Omron CX-Programmer project NewProject (CX-Programmer 9.73)

# PLC NewPLC1: CP1L-E EM

## Global symbols (name address type ; comment)
0.01 BOOL  ; SILINDER MAX (DISTRIBUTION)
0.04 BOOL  ; LIMIT SWITCH KIRI (DISTRIBUTION)
0.05 BOOL  ; LIMIT SWITCH KANAN (DISTRIBUTION)
0.06 BOOL  ; SENSOR BENDA (DISTRIBUTION)
100.00 BOOL  ; SOLENOID (DISTRIBUTION)
100.01 BOOL  ; SUCKER (DISTRIBUTION)
100.02 BOOL  ; BLOW (DISTRIBUTION)
100.03 BOOL  ; MOTOR KIRI (DISTRIBUTION)
100.04 BOOL  ; MOTOR KANAN (DISTRIBUTION)
101.00 BOOL  ; MOTOR KIRI (HANDLING)
101.01 BOOL  ; MOTOR KANAN (HANDLING)
101.02 BOOL  ; SOLENOID (HANDLING)
101.03 BOOL  ; GRAPLE (HANDLING)
101.04 BOOL  ; GRAPLE (HANDLING)
101.07 BOOL  ; TIDAK KIRIM DATA
1.00 BOOL  ; SENSOR BENDA AWAL (HANDLING)
1.01 BOOL  ; LIMIT SWITCH KIRI (HANDLING)
1.02 BOOL  ; LIMIT SWITCH KANAN (HANDLING)
1.03 BOOL  ; LIMIT SWITCH TENGAH (HANDLING)
1.04 BOOL  ; SILINDER MAX (HANDLING)
1.05 BOOL  ; SILINDER MIN (HANDLING)
1.06 BOOL  ; SENSOR BENDA GRAPLE (HANDLING)
W0.00 BOOL  ; START
W0.01 BOOL  ; STOP
W0.02 BOOL  ; RESET
W0.03 BOOL  ; SELECTOR SWITCH

## Program NewProgram1 (cyclic task 0)

### Section CONTROL

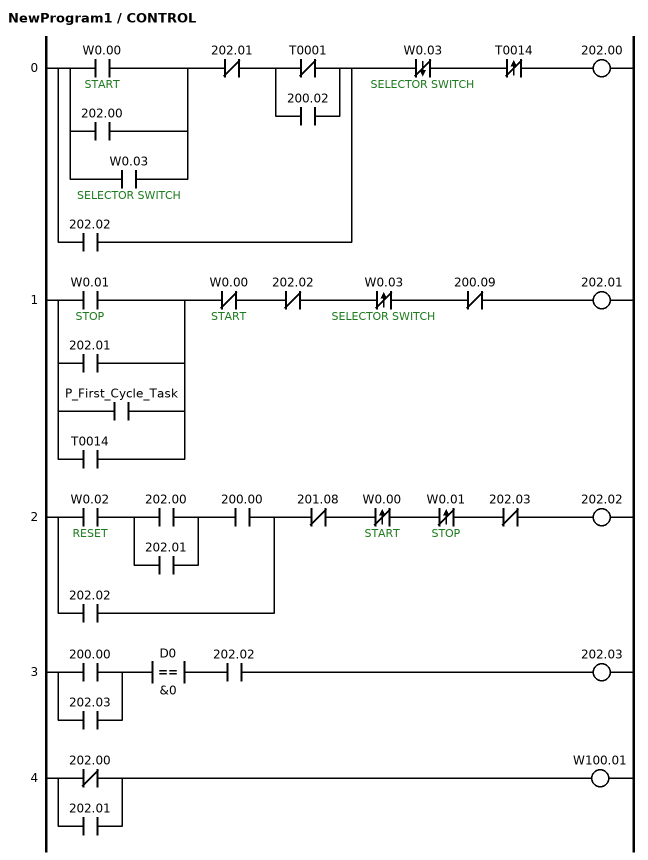
; rung 0
LD W0.00  ; START
OR 202.00
OR W0.03  ; SELECTOR SWITCH
ANDNOT 202.01
LDNOT T0001
OR 200.02
ANDLD
OR 202.02
%ANDNOT W0.03  ; SELECTOR SWITCH
@ANDNOT T0014
OUT 202.00
; rung 1
LD W0.01  ; STOP
OR 202.01
OR P_First_Cycle_Task
OR T0014
ANDNOT W0.00  ; START
ANDNOT 202.02
@ANDNOT W0.03  ; SELECTOR SWITCH
ANDNOT 200.09
OUT 202.01
; rung 2
LD W0.02  ; RESET
LD 202.00
OR 202.01
ANDLD
AND 200.00
OR 202.02
ANDNOT 201.08
@ANDNOT W0.00  ; START
@ANDNOT W0.01  ; STOP
ANDNOT 202.03
OUT 202.02
; rung 3
LD 200.00
OR 202.03
AND=(300) D0 &0
AND 202.02
OUT 202.03
; rung 4
LDNOT 202.00
OR 202.01
OUT W100.01

### Section DISTRIBUTION

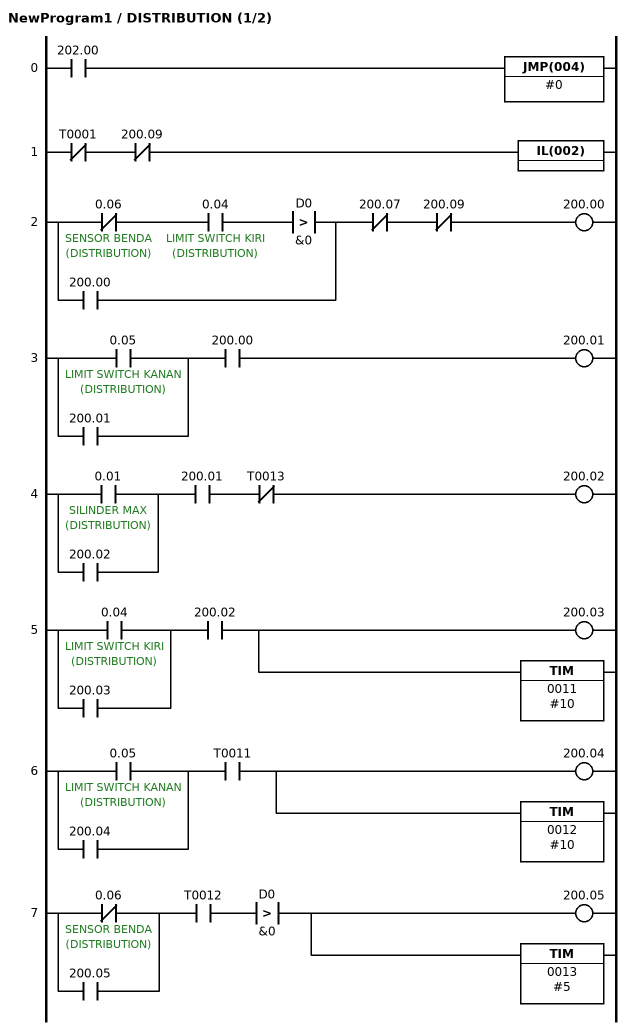
; rung 0
LD 202.00
JMP(004) #0
; rung 1
LDNOT T0001
ANDNOT 200.09
IL(002)
; rung 2
LDNOT 0.06  ; SENSOR BENDA (DISTRIBUTION)
AND 0.04  ; LIMIT SWITCH KIRI (DISTRIBUTION)
AND>(320) D0 &0
OR 200.00
ANDNOT 200.07
ANDNOT 200.09
OUT 200.00
; rung 3
LD 0.05  ; LIMIT SWITCH KANAN (DISTRIBUTION)
OR 200.01
AND 200.00
OUT 200.01
; rung 4
LD 0.01  ; SILINDER MAX (DISTRIBUTION)
OR 200.02
AND 200.01
ANDNOT T0013
OUT 200.02
; rung 5
LD 0.04  ; LIMIT SWITCH KIRI (DISTRIBUTION)
OR 200.03
AND 200.02
OUT 200.03
TIM 0011 #10
; rung 6
LD 0.05  ; LIMIT SWITCH KANAN (DISTRIBUTION)
OR 200.04
AND T0011
OUT 200.04
TIM 0012 #10
; rung 7
LDNOT 0.06  ; SENSOR BENDA (DISTRIBUTION)
OR 200.05
AND T0012
AND>(320) D0 &0
OUT 200.05
TIM 0013 #5

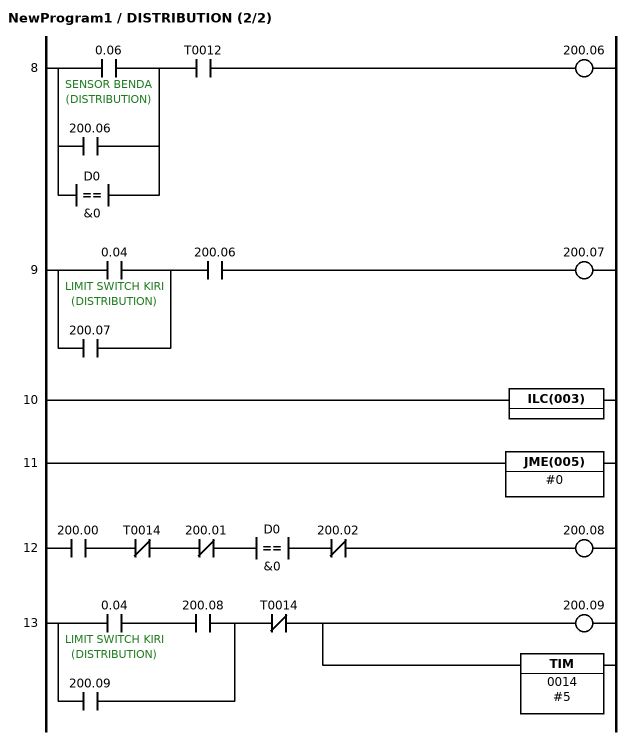
; rung 8
LD 0.06  ; SENSOR BENDA (DISTRIBUTION)
OR 200.06
OR=(300) D0 &0
AND T0012
OUT 200.06
; rung 9
LD 0.04  ; LIMIT SWITCH KIRI (DISTRIBUTION)
OR 200.07
AND 200.06
OUT 200.07
; rung 10
ILC(003)
; rung 11
JME(005) #0
; rung 12
LD 200.00
ANDNOT T0014
ANDNOT 200.01
AND=(300) D0 &0
ANDNOT 200.02
OUT 200.08
; rung 13
LD 0.04  ; LIMIT SWITCH KIRI (DISTRIBUTION)
AND 200.08
OR 200.09
ANDNOT T0014
OUT 200.09
TIM 0014 #5

### Section HANDLING

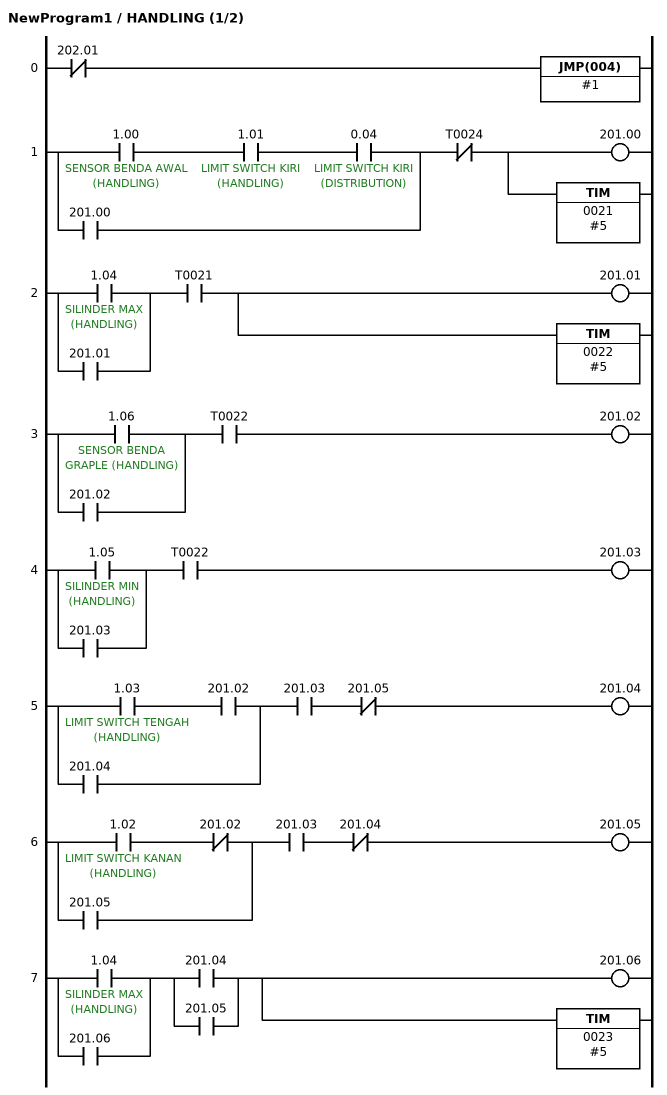
; rung 0
LDNOT 202.01
JMP(004) #1
; rung 1
LD 1.00  ; SENSOR BENDA AWAL (HANDLING)
AND 1.01  ; LIMIT SWITCH KIRI (HANDLING)
AND 0.04  ; LIMIT SWITCH KIRI (DISTRIBUTION)
OR 201.00
ANDNOT T0024
OUT 201.00
TIM 0021 #5
; rung 2
LD 1.04  ; SILINDER MAX (HANDLING)
OR 201.01
AND T0021
OUT 201.01
TIM 0022 #5
; rung 3
LD 1.06  ; SENSOR BENDA GRAPLE (HANDLING)
OR 201.02
AND T0022
OUT 201.02
; rung 4
LD 1.05  ; SILINDER MIN (HANDLING)
OR 201.03
AND T0022
OUT 201.03
; rung 5
LD 1.03  ; LIMIT SWITCH TENGAH (HANDLING)
AND 201.02
OR 201.04
AND 201.03
ANDNOT 201.05
OUT 201.04
; rung 6
LD 1.02  ; LIMIT SWITCH KANAN (HANDLING)
ANDNOT 201.02
OR 201.05
AND 201.03
ANDNOT 201.04
OUT 201.05
; rung 7
LD 1.04  ; SILINDER MAX (HANDLING)
OR 201.06
LD 201.04
OR 201.05
ANDLD
OUT 201.06
TIM 0023 #5

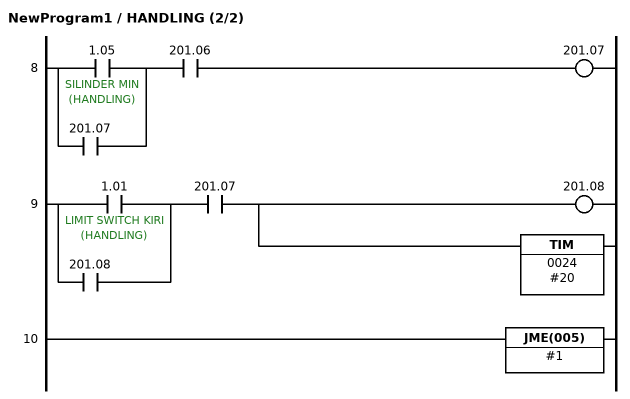
; rung 8
LD 1.05  ; SILINDER MIN (HANDLING)
OR 201.07
AND 201.06
OUT 201.07
; rung 9
LD 1.01  ; LIMIT SWITCH KIRI (HANDLING)
OR 201.08
AND 201.07
OUT 201.08
TIM 0024 #20
; rung 10
JME(005) #1

### Section OUTPUT

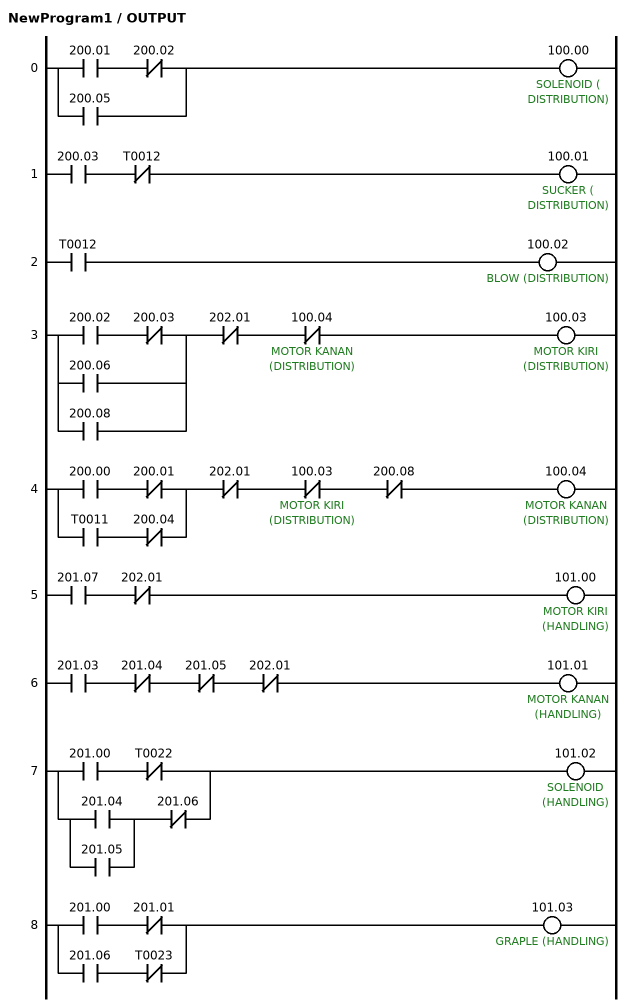
; rung 0
LD 200.01
ANDNOT 200.02
OR 200.05
OUT 100.00  ; SOLENOID (DISTRIBUTION)
; rung 1
LD 200.03
ANDNOT T0012
OUT 100.01  ; SUCKER (DISTRIBUTION)
; rung 2
LD T0012
OUT 100.02  ; BLOW (DISTRIBUTION)
; rung 3
LD 200.02
ANDNOT 200.03
OR 200.06
OR 200.08
ANDNOT 202.01
ANDNOT 100.04  ; MOTOR KANAN (DISTRIBUTION)
OUT 100.03  ; MOTOR KIRI (DISTRIBUTION)
; rung 4
LD 200.00
ANDNOT 200.01
LD T0011
ANDNOT 200.04
ORLD
ANDNOT 202.01
ANDNOT 100.03  ; MOTOR KIRI (DISTRIBUTION)
ANDNOT 200.08
OUT 100.04  ; MOTOR KANAN (DISTRIBUTION)
; rung 5
LD 201.07
ANDNOT 202.01
OUT 101.00  ; MOTOR KIRI (HANDLING)
; rung 6
LD 201.03
ANDNOT 201.04
ANDNOT 201.05
ANDNOT 202.01
OUT 101.01  ; MOTOR KANAN (HANDLING)
; rung 7
LD 201.00
ANDNOT T0022
LD 201.04
OR 201.05
ANDNOT 201.06
ORLD
OUT 101.02  ; SOLENOID (HANDLING)
; rung 8
LD 201.00
ANDNOT 201.01
LD 201.06
ANDNOT T0023
ORLD
OUT 101.03  ; GRAPLE (HANDLING)

### Section DATA_DISTRIBUTION

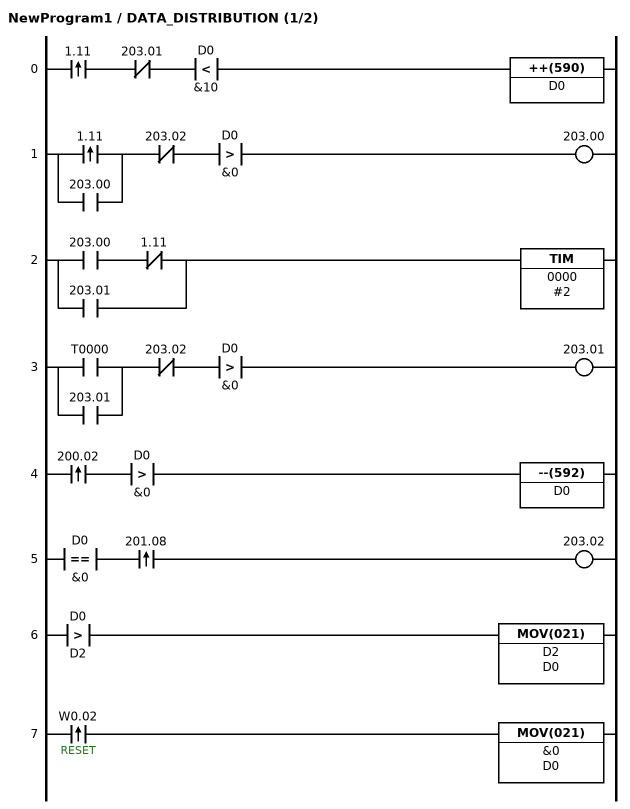
; rung 0
@LD 1.11
ANDNOT 203.01
AND<(310) D0 &10
++(590) D0
; rung 1
@LD 1.11
OR 203.00
ANDNOT 203.02
AND>(320) D0 &0
OUT 203.00
; rung 2
LD 203.00
ANDNOT 1.11
OR 203.01
TIM 0000 #2
; rung 3
LD T0000
OR 203.01
ANDNOT 203.02
AND>(320) D0 &0
OUT 203.01
; rung 4
@LD 200.02
AND>(320) D0 &0
--(592) D0
; rung 5
LD=(300) D0 &0
@AND 201.08
OUT 203.02
; rung 6
LD>(320) D0 D2
MOV(021) D2 D0
; rung 7
@LD W0.02  ; RESET
MOV(021) &0 D0

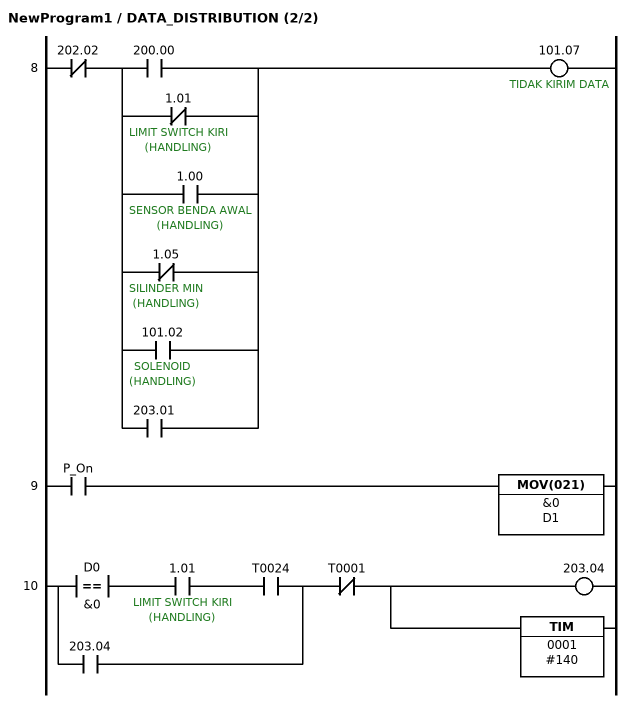
; rung 8
LDNOT 202.02
LD 200.00
ORNOT 1.01  ; LIMIT SWITCH KIRI (HANDLING)
OR 1.00  ; SENSOR BENDA AWAL (HANDLING)
ORNOT 1.05  ; SILINDER MIN (HANDLING)
OR 101.02  ; SOLENOID (HANDLING)
OR 203.01
ANDLD
OUT 101.07  ; TIDAK KIRIM DATA
; rung 9
LD P_On
MOV(021) &0 D1
; rung 10
LD=(300) D0 &0
AND 1.01  ; LIMIT SWITCH KIRI (HANDLING)
AND T0024
OR 203.04
ANDNOT T0001
OUT 203.04
TIM 0001 #140

### Section END
; rung 0
END(001)